# EPICS substitutions: bpmApp/Db/ai_xy_pos.substitutions
file ai_xy_pos.template
{ pattern
{CNO,       N, OFFSET_X, OFFSET_Y, LEN}
{ "\$(CNO)",  "\$(N)", "\$(OFFSET_X)", "\$(OFFSET_Y)", "\$(LEN)" }
}
